// Mitsubishi GX Works2 project: automation   PLC: FX3G

// global labels: Global1
VAR_GLOBAL
  start_flavor_prep AT X001 : BOOL;
  start_cooling AT X002 : BOOL;
  temp_sensor AT X003 : BOOL;
  emergency_button AT X005 : BOOL;
  start_day_button AT X007 : BOOL;
  flavor_prep_light AT Y000 : BOOL;
  cooling_light AT Y002 : BOOL;
  blink_y5 AT Y005 : BOOL;
  blink_y6 AT Y006 : BOOL;
  day_active AT Y007 : BOOL;
  day_end AT M10 : BOOL;
  move_quantity AT M50 : BOOL;
  normalized_input AT M65 : BOOL;
  Regular AT M70 : BOOL;
  Premium AT M75 : BOOL;
  cant_produce AT M80 : BOOL;
  mixing_done AT M90 : BOOL;
  raspberry_input AT D1100 : REAL;
  lemon_input AT D1110 : REAL;
  stabilizer_input AT D1120 : REAL;
  gummies_input AT D1130 : REAL;
  raspberry_quantity AT D1200 : REAL;
  lemon_quantity AT D1210 : REAL;
  stabilizer_quantity AT D1220 : REAL;
  gummies_quantity AT D1230 : REAL;
  raspberry_cooling_tank AT D1300 : REAL;
  lemon_cooling_tank AT D1310 : REAL;
  mix_tank AT D1400 : REAL;
  storage_tank AT D1500 : REAL;
  gummy_type AT D1600 : REAL;
  AnalogInput1 AT D8280 : INT;
  TC_flavor AT TC1 : BOOL;
  TC_cooling AT TC2 : BOOL;
  TC_mix_regular AT TC3 : BOOL;
  TC_mix_premium AT TC4 : BOOL;
  stop_flavor AT TS1 : BOOL;
  stop_cooling AT TS2 : BOOL;
  stop_mix_regular AT TS3 : BOOL;
  stop_mix_premium AT TS4 : BOOL;
END_VAR
VAR_GLOBAL CONSTANT
  constant_0 : REAL;
  constant_400 : REAL := 400.0;
  constant_5 : REAL := 5.0;
  constant_10 : INT := 10;
  constant_280 : REAL := 280.0;
  constant_105 : REAL := 105.0;
  constant_455 : REAL := 455.0;
  constant_28 : REAL := 28.0;
  constant_385 : REAL := 385.0;
  constant_665 : REAL := 665.0;
  constant_210 : REAL := 210.0;
  constant_70 : REAL := 70.0;
  constant_350 : REAL := 350.0;
  constant_490 : REAL := 490.0;
  constant_560 : REAL := 560.0;
  constant_700 : REAL := 700.0;
  constant_50 : INT := 50;
  constant_80 : INT := 80;
  constant_30 : INT := 30;
  constant_1 : REAL := 1.0;
  constant_10_float : REAL := 10.0;
  constant_zero : INT;
END_VAR
VAR_GLOBAL
  raspberry_prep_tank AT D1150 : REAL;
  lemon_prep_tank AT D1160 : REAL;
  mix_trigger AT M100 : BOOL;
END_VAR
VAR_GLOBAL CONSTANT
  constant_530 : INT := 50;
END_VAR
VAR_GLOBAL
  Blink_help AT M500 : BOOL;
  TC_Blinker_1 AT TC5 : BOOL;
  TC_Blinker_2 AT TC6 : BOOL;
  TS_Stop_Blinker_1 AT TS5 : BOOL;
  TS_Stop_Blinker_2 AT TS6 : BOOL;
  Finished_cool AT M120 : BOOL;
END_VAR
VAR_GLOBAL CONSTANT
  constant_386 : REAL := 386.0;
  constant_666 : REAL := 666.0;
  constant_211 : REAL := 211.0;
  constant_71 : REAL := 71.0;
  constant_281 : REAL := 281;
END_VAR
VAR_GLOBAL
  temp_analog_val AT D1180 : REAL;
  Analog_output AT D8282 : INT;
END_VAR
VAR_GLOBAL CONSTANT
  constant_40 : REAL := 40;
END_VAR

// task Task_01 (event TRUE, interval 0, priority 31): POU_01

PROGRAM POU_01
(* structured ladder/FBD written out as ST: instructions are called as NAME(EN, inputs, outputs); _pN, _eN, _tN stand for wires *)
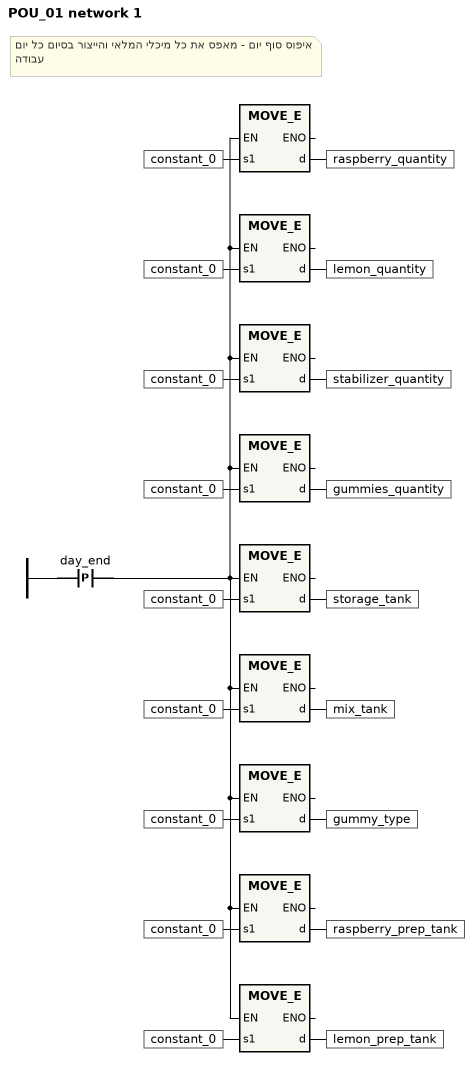
(* network 1 *)
(* איפוס סוף יום - מאפס את כל מיכלי המלאי והייצור בסיום כל יום עבודה *)
_p1 := LDP(TRUE, day_end);
MOVE_E(_p1, constant_0, raspberry_quantity);
MOVE_E(_p1, constant_0, lemon_quantity);
MOVE_E(_p1, constant_0, stabilizer_quantity);
MOVE_E(_p1, constant_0, gummies_quantity);
MOVE_E(_p1, constant_0, storage_tank);
MOVE_E(_p1, constant_0, mix_tank);
MOVE_E(_p1, constant_0, gummy_type);
MOVE_E(_p1, constant_0, raspberry_prep_tank);
MOVE_E(_p1, constant_0, lemon_prep_tank);
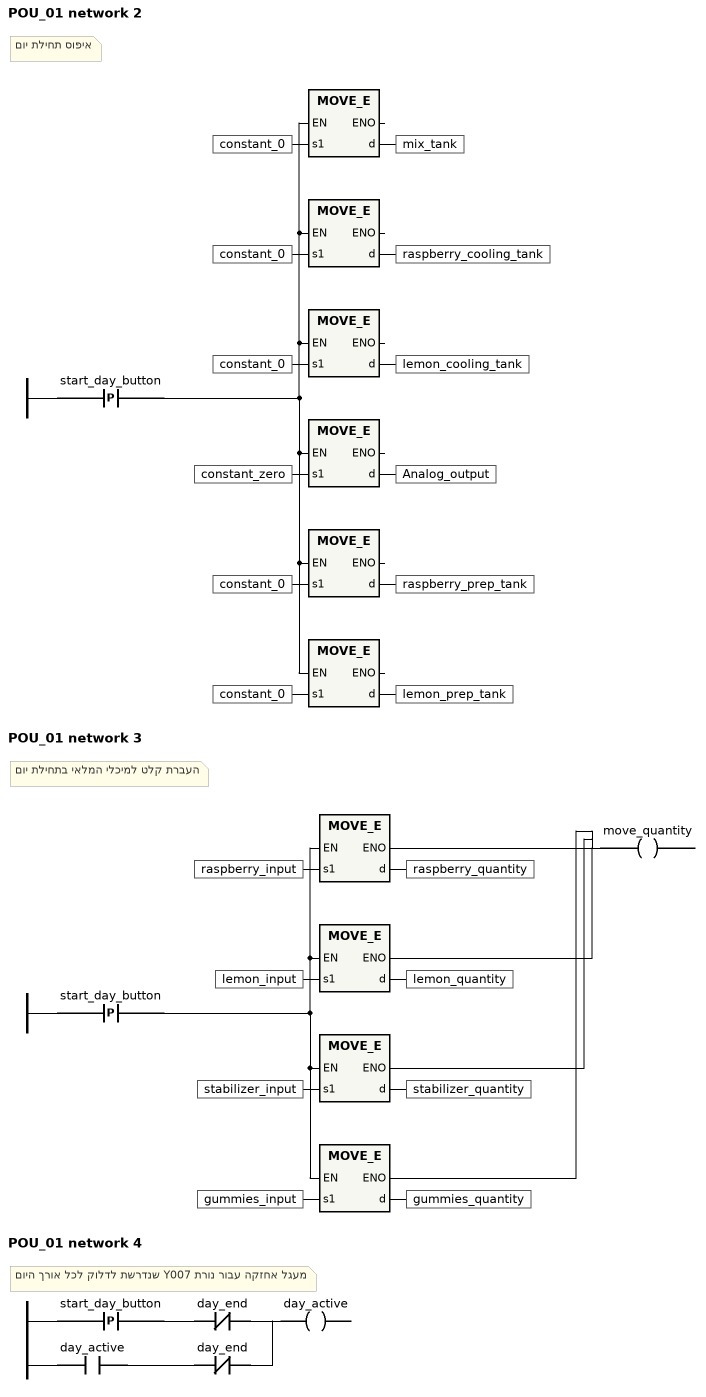
(* network 2 *)
(* איפוס תחילת יום *)
_p1 := LDP(TRUE, start_day_button);
MOVE_E(_p1, constant_0, mix_tank);
MOVE_E(_p1, constant_0, raspberry_cooling_tank);
MOVE_E(_p1, constant_0, lemon_cooling_tank);
MOVE_E(_p1, constant_zero, Analog_output);
MOVE_E(_p1, constant_0, raspberry_prep_tank);
MOVE_E(_p1, constant_0, lemon_prep_tank);
(* network 3 *)
(* העברת קלט למיכלי המלאי בתחילת יום *)
_p1 := LDP(TRUE, start_day_button);
_e2 := MOVE_E(_p1, raspberry_input, raspberry_quantity);
_e3 := MOVE_E(_p1, lemon_input, lemon_quantity);
_e4 := MOVE_E(_p1, stabilizer_input, stabilizer_quantity);
_e5 := MOVE_E(_p1, gummies_input, gummies_quantity);
move_quantity := _e2 OR _e3 OR _e4 OR _e5;
(* network 4 *)
(* מעגל אחזקה עבור נורת Y007 שנדרשת לדלוק לכל אורך היום *)
day_active := (LDP(TRUE, start_day_button) AND NOT day_end) OR (day_active AND NOT day_end);
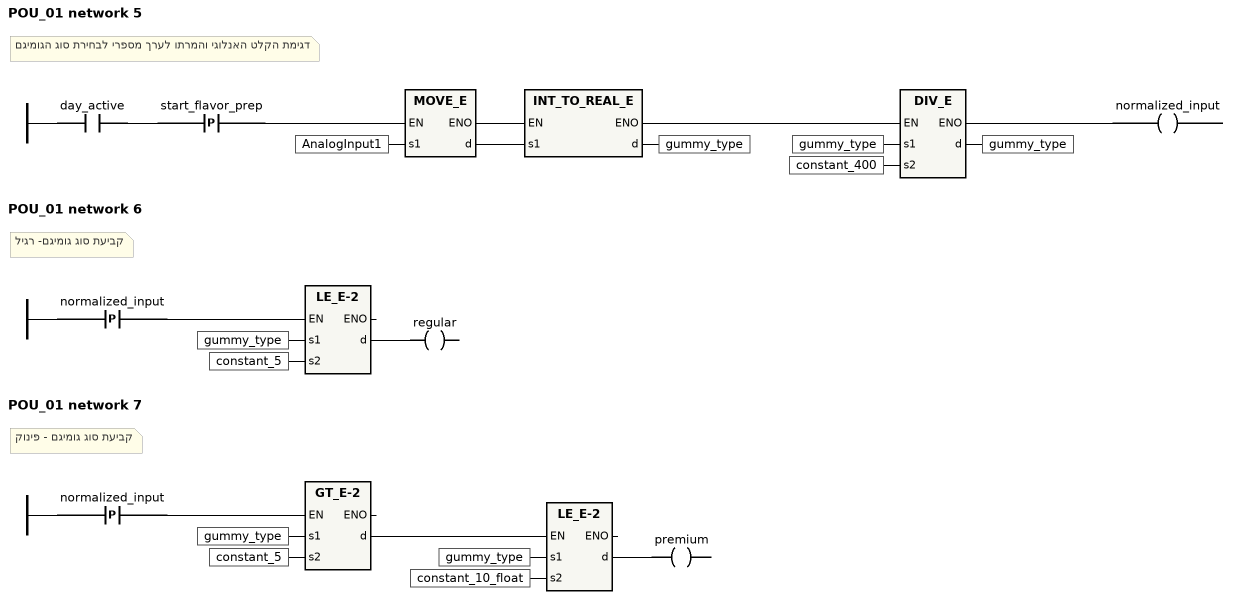
(* network 5 *)
(* דגימת הקלט האנלוגי והמרתו לערך מספרי לבחירת סוג הגומיגם *)
_e2 := MOVE_E(day_active AND LDP(TRUE, start_flavor_prep), AnalogInput1, _t1);
_e3 := INT_TO_REAL_E(_e2, _t1, gummy_type);
_e4 := DIV_E(_e3, gummy_type, constant_400, gummy_type);
normalized_input := _e4;
(* network 6 *)
(* קביעת סוג גומיגם- רגיל *)
LE_E(LDP(TRUE, normalized_input), gummy_type, constant_5, _t1);
regular := _t1;
(* network 7 *)
(* קביעת סוג גומיגם - פינוק *)
GT_E(LDP(TRUE, normalized_input), gummy_type, constant_5, _t1);
LE_E(_t1, gummy_type, constant_10_float, _t2);
premium := _t2;
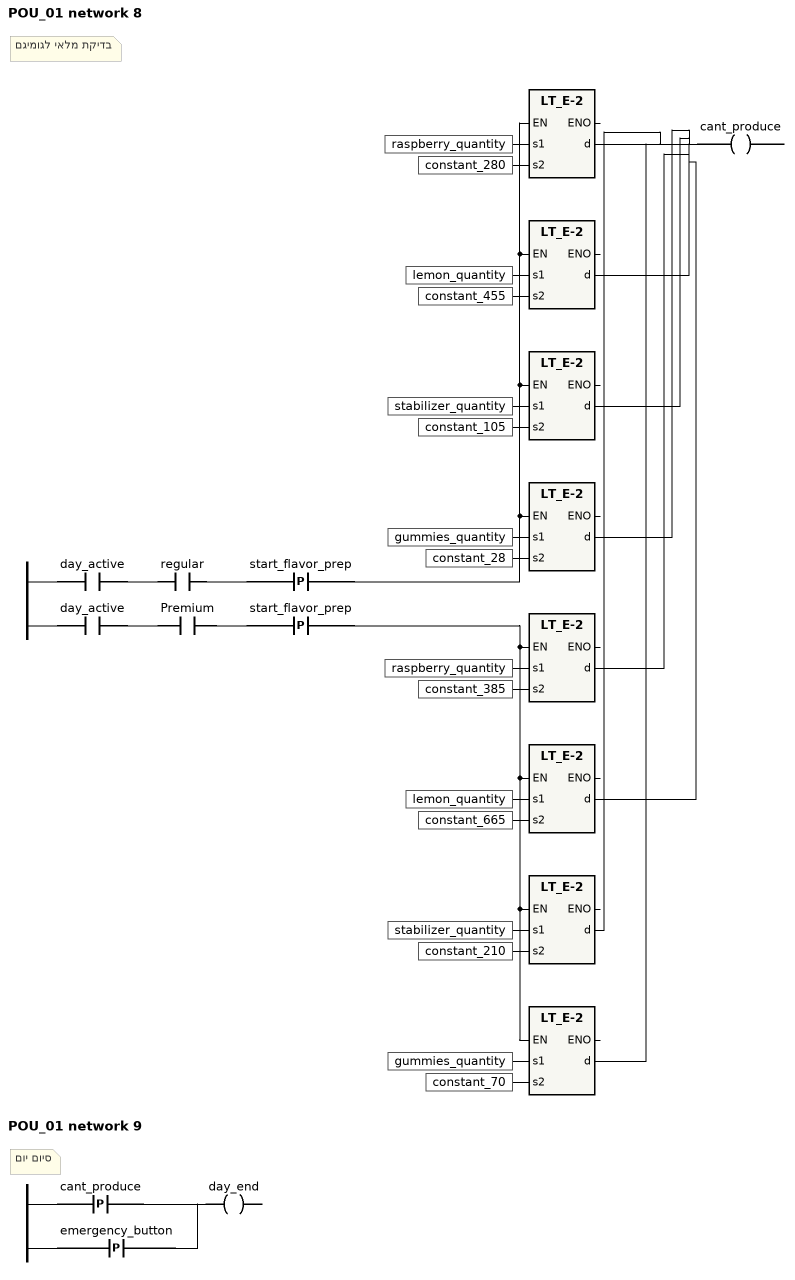
(* network 8 *)
(* בדיקת מלאי לגומיגם *)
_p1 := day_active AND regular AND LDP(TRUE, start_flavor_prep);
LT_E(_p1, raspberry_quantity, constant_280, _t2);
LT_E(_p1, lemon_quantity, constant_455, _t3);
LT_E(_p1, stabilizer_quantity, constant_105, _t4);
LT_E(_p1, gummies_quantity, constant_28, _t5);
_p6 := day_active AND Premium AND LDP(TRUE, start_flavor_prep);
LT_E(_p6, raspberry_quantity, constant_385, _t7);
LT_E(_p6, lemon_quantity, constant_665, _t8);
LT_E(_p6, stabilizer_quantity, constant_210, _t9);
LT_E(_p6, gummies_quantity, constant_70, _t10);
cant_produce := _t2 OR _t3 OR _t4 OR _t5 OR _t7 OR _t8 OR _t9 OR _t10;
(* network 9 *)
(* סיום יום *)
day_end := LDP(TRUE, cant_produce) OR LDP(TRUE, emergency_button);
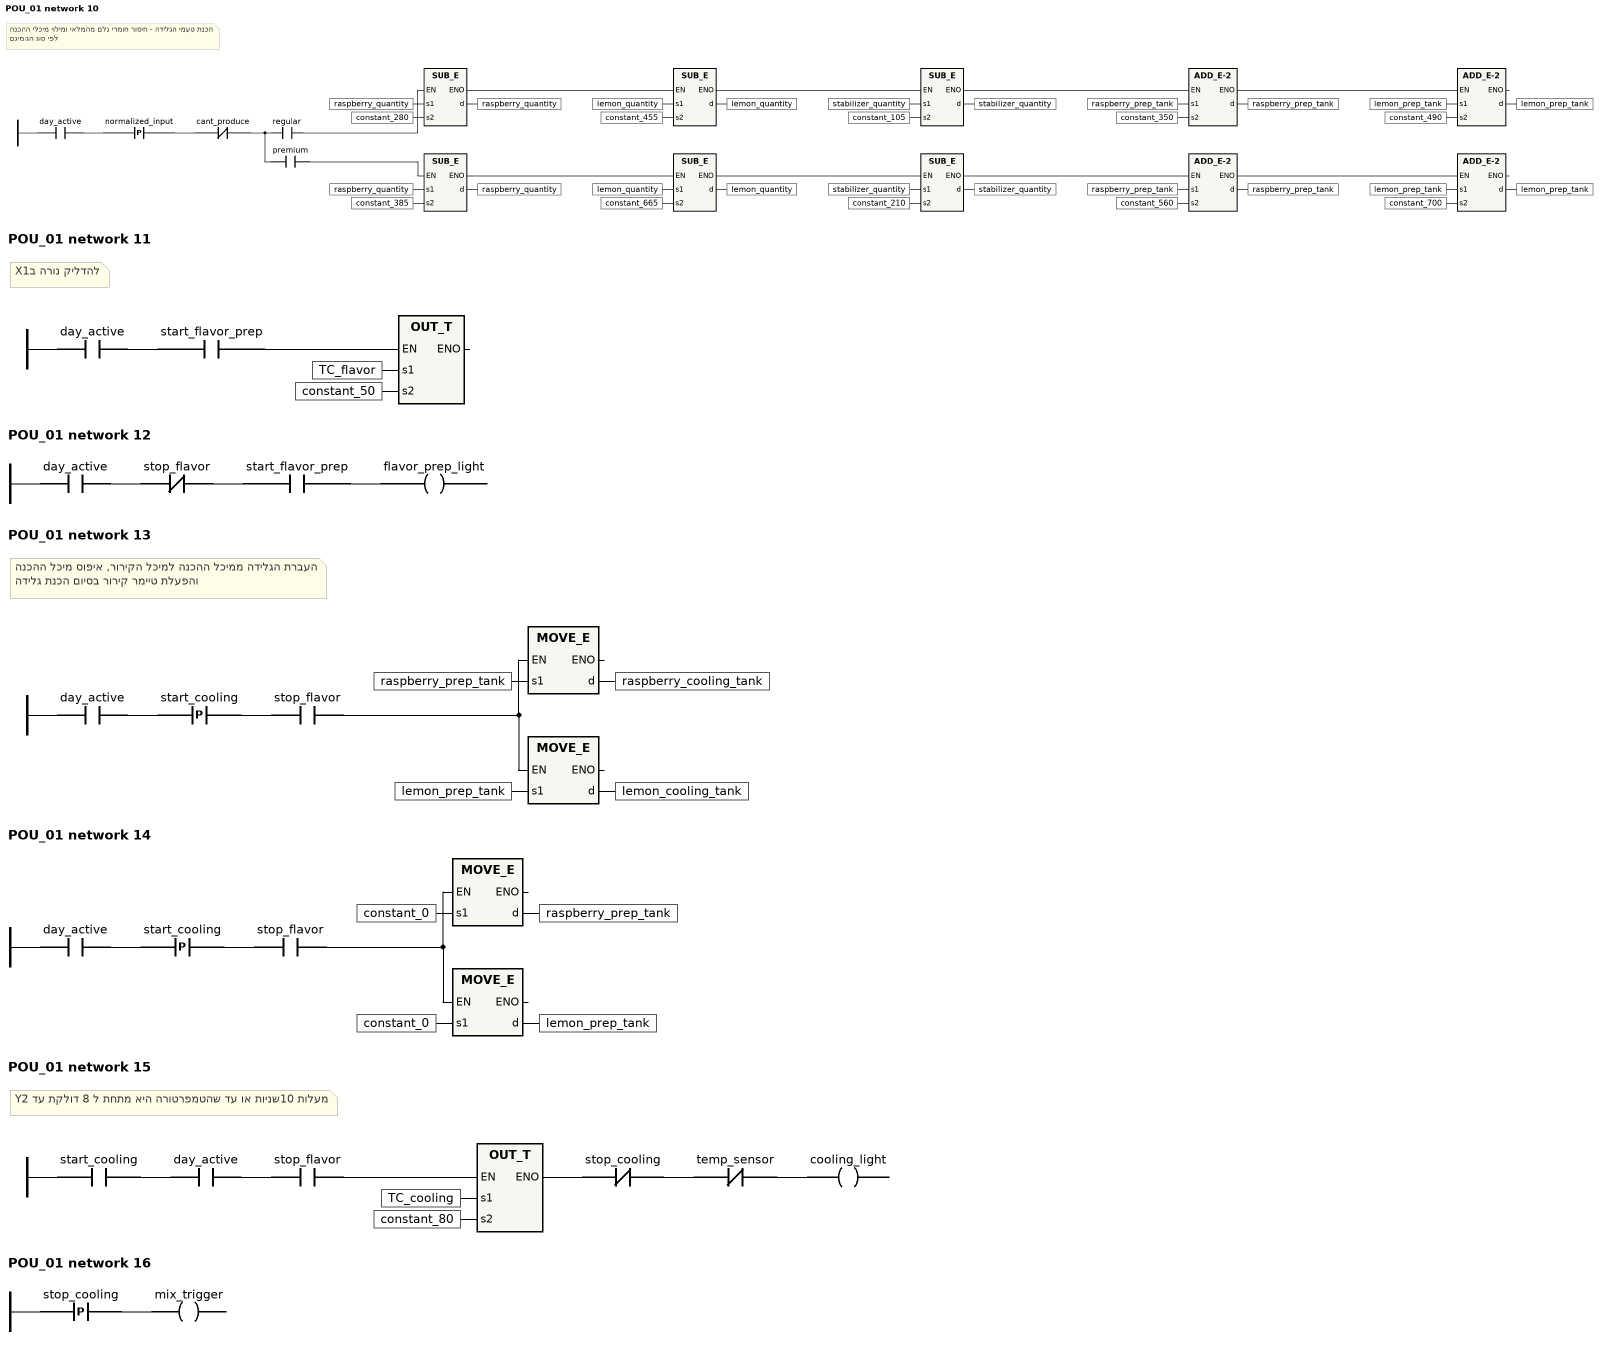
(* network 10 *)
(* הכנת טעמי הגלידה - חיסור חומרי גלם מהמלאי ומילוי מיכלי ההכנה לפי סוג הגומיגם *)
_p1 := day_active AND LDP(TRUE, normalized_input) AND NOT cant_produce;
_e2 := SUB_E(_p1 AND regular, raspberry_quantity, constant_280, raspberry_quantity);
_e3 := SUB_E(_e2, lemon_quantity, constant_455, lemon_quantity);
_e4 := SUB_E(_e3, stabilizer_quantity, constant_105, stabilizer_quantity);
_e5 := ADD_E(_e4, raspberry_prep_tank, constant_350, raspberry_prep_tank);
ADD_E(_e5, lemon_prep_tank, constant_490, lemon_prep_tank);
_e6 := SUB_E(_p1 AND premium, raspberry_quantity, constant_385, raspberry_quantity);
_e7 := SUB_E(_e6, lemon_quantity, constant_665, lemon_quantity);
_e8 := SUB_E(_e7, stabilizer_quantity, constant_210, stabilizer_quantity);
_e9 := ADD_E(_e8, raspberry_prep_tank, constant_560, raspberry_prep_tank);
ADD_E(_e9, lemon_prep_tank, constant_700, lemon_prep_tank);
(* network 11 *)
(* להדליק נורה בX1 *)
OUT_T(day_active AND start_flavor_prep, TC_flavor, constant_50);
(* network 12 *)
flavor_prep_light := day_active AND NOT stop_flavor AND start_flavor_prep;
(* network 13 *)
(* העברת הגלידה ממיכל ההכנה למיכל הקירור, איפוס מיכל ההכנה והפעלת טיימר קירור בסיום הכנת גלידה *)
_p1 := day_active AND LDP(TRUE, start_cooling) AND stop_flavor;
MOVE_E(_p1, raspberry_prep_tank, raspberry_cooling_tank);
MOVE_E(_p1, lemon_prep_tank, lemon_cooling_tank);
(* network 14 *)
_p1 := day_active AND LDP(TRUE, start_cooling) AND stop_flavor;
MOVE_E(_p1, constant_0, raspberry_prep_tank);
MOVE_E(_p1, constant_0, lemon_prep_tank);
(* network 15 *)
(* Y2 דולקת עד 8 שניות או עד שהטמפרטורה היא מתחת ל10 מעלות *)
_e1 := OUT_T(start_cooling AND day_active AND stop_flavor, TC_cooling, constant_80);
cooling_light := _e1 AND NOT stop_cooling AND NOT temp_sensor;
(* network 16 *)
mix_trigger := LDP(TRUE, stop_cooling);
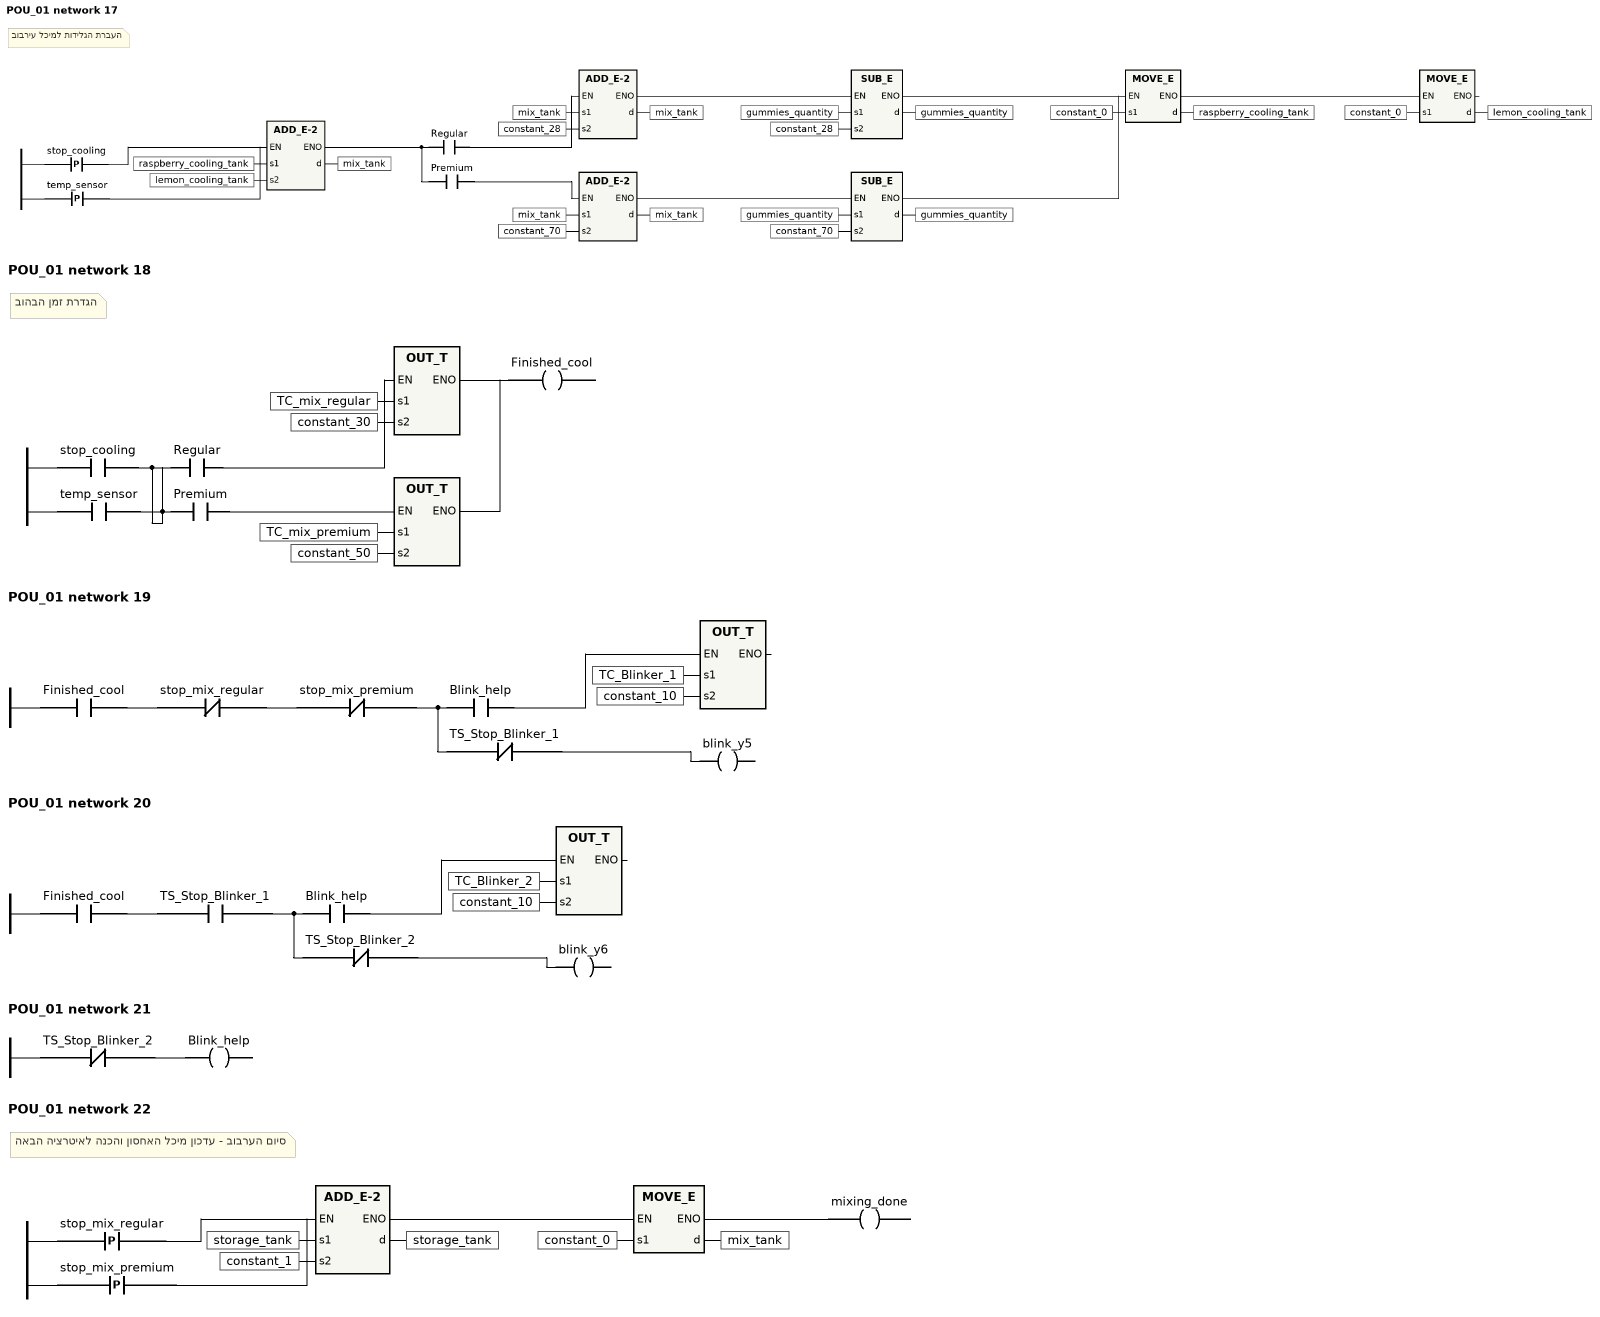
(* network 17 *)
(* העברת הגלידות למיכל עירבוב *)
_e1 := ADD_E(LDP(TRUE, stop_cooling) OR LDP(TRUE, temp_sensor), raspberry_cooling_tank, lemon_cooling_tank, mix_tank);
_e2 := ADD_E(_e1 AND Regular, mix_tank, constant_28, mix_tank);
_e3 := SUB_E(_e2, gummies_quantity, constant_28, gummies_quantity);
_e4 := ADD_E(_e1 AND Premium, mix_tank, constant_70, mix_tank);
_e5 := SUB_E(_e4, gummies_quantity, constant_70, gummies_quantity);
_e6 := MOVE_E(_e3 OR _e5, constant_0, raspberry_cooling_tank);
MOVE_E(_e6, constant_0, lemon_cooling_tank);
(* network 18 *)
(* הגדרת זמן הבהוב *)
_p1 := stop_cooling OR temp_sensor;
_e2 := OUT_T(_p1 AND Regular, TC_mix_regular, constant_30);
_e3 := OUT_T(_p1 AND Premium, TC_mix_premium, constant_50);
Finished_cool := _e2 OR _e3;
(* network 19 *)
_p1 := Finished_cool AND NOT stop_mix_regular AND NOT stop_mix_premium;
OUT_T(_p1 AND Blink_help, TC_Blinker_1, constant_10);
blink_y5 := _p1 AND NOT TS_Stop_Blinker_1;
(* network 20 *)
_p1 := Finished_cool AND TS_Stop_Blinker_1;
OUT_T(_p1 AND Blink_help, TC_Blinker_2, constant_10);
blink_y6 := _p1 AND NOT TS_Stop_Blinker_2;
(* network 21 *)
Blink_help := NOT TS_Stop_Blinker_2;
(* network 22 *)
(* סיום הערבוב - עדכון מיכל האחסון והכנה לאיטרציה הבאה *)
_e1 := ADD_E(LDP(TRUE, stop_mix_regular) OR LDP(TRUE, stop_mix_premium), storage_tank, constant_1, storage_tank);
_e2 := MOVE_E(_e1, constant_0, mix_tank);
mixing_done := _e2;
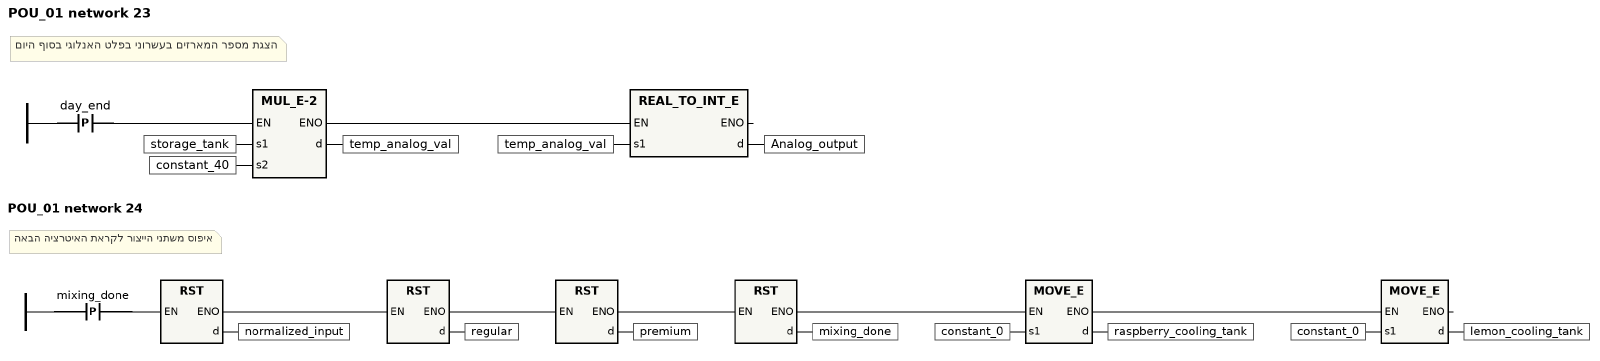
(* network 23 *)
(* הצגת מספר המארזים בעשרוני בפלט האנלוגי בסוף היום *)
_e1 := MUL_E(LDP(TRUE, day_end), storage_tank, constant_40, temp_analog_val);
REAL_TO_INT_E(_e1, temp_analog_val, Analog_output);
(* network 24 *)
(* איפוס משתני הייצור לקראת האיטרציה הבאה *)
_e1 := RST(LDP(TRUE, mixing_done), normalized_input);
_e2 := RST(_e1, regular);
_e3 := RST(_e2, premium);
_e4 := RST(_e3, mixing_done);
_e5 := MOVE_E(_e4, constant_0, raspberry_cooling_tank);
MOVE_E(_e5, constant_0, lemon_cooling_tank);
END_PROGRAM
